{attribute 'GeneratedUsingTerminal: EK1122-0000-0018'}
{attribute addProperty BoxType "EK1122-0000-0018"}
{attribute addProperty Id "RP20_VI_AES_D_BC_ECAT_xAES_B47A261080RP20_SAFETY_Flexi_Soft_EtherCAT_GatewayFlexi_Soft_EtherCAT_Gateway_DE394EDD5RP20_AB0_EPP1322_0001EPP1322_1FC0878B2RP20_AB1_EPP1008_0001EPP1008_78E8D3DD12RP20_AB2_EPP1008_0001EPP1008_78E8D3DD12RP20_AB3_EPP1008_0001EPP1008_78E8D3DD12RP20_AB4_EPP1008_0001EPP1008_78E8D3DD12"}
{attribute addProperty CRC "1758988522"}
{attribute addProperty Size "135"}
{attribute addProperty Name "RP20_A2 (EK1122)"}
TYPE RP20_A2_EK1122_68D808EA EXTENDS EK1122_1FC0878B :
STRUCT
	{attribute addProperty Name "RP20-VI (AES-D-BC-ECAT)"}
	{attribute addProperty PreviousPort "RP20_A2 (EK1122) : D"}
	RP20_VI_AES_D_BC_ECAT_x : AES_B47A2610;
	{attribute addProperty Name "RP20-SAFETY (Flexi Soft EtherCAT Gateway)"}
	{attribute addProperty PreviousPort "RP20_A2 (EK1122) : B"}
	RP20_SAFETY_Flexi_Soft_EtherCAT_Gateway : Flexi_Soft_EtherCAT_Gateway_DE394EDD;
	{attribute addProperty Name "RP20-AB0 (EPP1322-0001)"}
	{attribute addProperty PreviousPort "RP20-SAFETY (Flexi Soft EtherCAT Gateway) : B"}
	RP20_AB0_EPP1322_0001 : EPP1322_1FC0878B;
	{attribute addProperty Name "RP20-AB1 (EPP1008-0001)"}
	{attribute addProperty PreviousPort "RP20-AB0 (EPP1322-0001) : C"}
	RP20_AB1_EPP1008_0001 : EPP1008_78E8D3DD;
	{attribute addProperty Name "RP20-AB2 (EPP1008-0001)"}
	{attribute addProperty PreviousPort "RP20-AB1 (EPP1008-0001) : B"}
	RP20_AB2_EPP1008_0001 : EPP1008_78E8D3DD;
	{attribute addProperty Name "RP20-AB3 (EPP1008-0001)"}
	{attribute addProperty PreviousPort "RP20-AB2 (EPP1008-0001) : B"}
	RP20_AB3_EPP1008_0001 : EPP1008_78E8D3DD;
	{attribute addProperty Name "RP20-AB4 (EPP1008-0001)"}
	{attribute addProperty PreviousPort "RP20-AB3 (EPP1008-0001) : B"}
	RP20_AB4_EPP1008_0001 : EPP1008_78E8D3DD;
END_STRUCT
END_TYPE

(* stored: Version 1.2.0.0, ProductVersion 3.1.4024.11
   DUT RP20_A2_EK1122_68D808EA: Id {f776b7ef-d479-08b0-3215-082da0c90041} *)
